// TwinCAT 3 PLC project Untitled1
// ProgramVersion: 3.1.4024.12
// libraries:
//   Tc2_Standard, * (Beckhoff Automation GmbH)
//   Tc2_System, * (Beckhoff Automation GmbH)
//   Tc3_Module, * (Beckhoff Automation GmbH)
// project tree:
//   Loadstation/ Parts.TcGVL, MAIN.TcPOU
//   Loadstation/State_Command_Enum/ Command.TcDUT, DUT.TcTLEO
//   / PlcTask.TcTTO
//   Loadstation/2_Control/ CON_LoadingStation.TcPOU
//   Loadstation/2_Control/Loadingstation/DataTypes/ MOD_Loadingstation_I_stWeighbridge.TcDUT (not stored), MOD_Loadingstation_Q_stCrane.TcDUT
//   Loadstation/3_Module/Crane/DataTypes/ MOD_Crane_I_stLoad.TcDUT, MOD_Crane_I_stSensor.TcDUT (not stored), MOD_Crane_Q_stMotor.TcDUT (not stored)
//   Loadstation/3_Module/Crane/ MOD_Crane.TcPOU
//   Loadstation/3_Module/InputBelt/DataTypes/ MOD_InputBelt_I_stSensor.TcDUT (not stored), MOD_InputBelt_Q_stMotor.TcDUT (not stored), MOD_InputBelt_Q_stOutput.TcDUT, MOD_InputBelt_Q_stRequest.TcDUT (not stored)
//   Loadstation/3_Module/InputBelt/ MOD_InputBelt.TcPOU
//   Loadstation/3_Module/ MOD_MechanicalGrabCrane.TcPOU (not stored)
//   Loadstation/3_Module/WeighBridge/DataTypes/ MOD_WeighBridge_I_stDefinitions.TcDUT, MOD_Weighbridge_I_stSensor.TcDUT (not stored), MOD_WeighBridge_Q_stOutput.TcDUT (not stored)
//   Loadstation/3_Module/WeighBridge/ MOD_Weighbridge.TcPOU
//   Loadstation/4_Devices/Motor_Notimplemented/Sensor/ DEV_Sensor_stOutput.TcDUT
//   Loadstation/4_Devices/ Motor_Notimplemented.TcPOU (not stored), Sensor_Notimplemented.TcPOU (not stored)
//   Loadstation/Application/ FB2_Control.TcPOU, FB3_Modules.TcPOU, FB4_Devices.TcPOU
// real-time tasks:
//   TASK PlcTask: cycle T#10ms, priority 20, ADS port 350

CONFIGURATION Untitled1
    RESOURCE PLC ON TwinCAT3
        TASK PlcTask(INTERVAL := T#10ms, PRIORITY := 20);
        PROGRAM MAIN WITH PlcTask : MAIN;
    END_RESOURCE
END_CONFIGURATION

// ---- Loadstation/State_Command_Enum/Command.TcDUT
{attribute 'qualified_only'}
{attribute 'strict'}
TYPE Command :
(
	Stop 		:= 0,
	Abort 		:= 1,
	Executing 	:= 2,
	Hold 		:= 3,
	Reset 		:= 4
);
END_TYPE

// ---- Loadstation/State_Command_Enum/DUT.TcTLEO
{attribute 'qualified_only'}
{attribute 'strict'}
TYPE DUT :
(
	Aborting := 0,
	Aborted		:= 1,
	
	Clearing	:= 2,
	Stopping	:= 3,
	Stopped		:= 4,
	
	Resetting	:= 5,
	Idle		:= 6,
	Starting	:= 7,
	Execute		:= 8,
	
	Holding		:= 9,
	Held		:= 10,
	Unholding		:= 11,
	
	Suspending		:= 12,
	Suspended		:= 13,
	Unsuspending	:= 14,
	
	Complete 		:= 15
);
END_TYPE

// ---- Loadstation/2_Control/Loadingstation/DataTypes/MOD_Loadingstation_Q_stCrane.TcDUT
TYPE MOD_Loadingstation_Q_stCrane :
STRUCT
	AllowedToOperate : BOOL;
END_STRUCT
END_TYPE

// ---- Loadstation/3_Module/Crane/DataTypes/MOD_Crane_I_stLoad.TcDUT
TYPE MOD_Crane_I_stLoad :
STRUCT
	Ready : BOOL;
	AllowedToOperate : BOOL;
END_STRUCT
END_TYPE

// ---- Loadstation/3_Module/InputBelt/DataTypes/MOD_InputBelt_Q_stOutput.TcDUT
TYPE MOD_InputBelt_Q_stOutput :
STRUCT
	BoxReady : BOOL;
END_STRUCT
END_TYPE

// ---- Loadstation/3_Module/WeighBridge/DataTypes/MOD_WeighBridge_I_stDefinitions.TcDUT
TYPE MOD_WeighBridge_I_stDefinitions :
STRUCT
	WeightLimit : INT;
	OperatingWeight : INT;
	DetractorWeight : INT;
END_STRUCT
END_TYPE

// ---- Loadstation/4_Devices/Motor_Notimplemented/Sensor/DEV_Sensor_stOutput.TcDUT
TYPE DEV_Sensor_stOutput :
STRUCT
	Abort : BOOL;
	Detecting : BOOL;
END_STRUCT
END_TYPE

// ---- Loadstation/Parts.TcGVL
//{attribute 'qualified_only'}
VAR_GLOBAL
	GlobalCommandState : INT;	

	//control
	Loadingstation : CON_LoadingStation; 
	
	//Modules
	Belt : MOD_InputBelt;
	Crane : MOD_Crane;
	Weighbridge : MOD_Weighbridge;
	MechanicalGrabCrane : MOD_MechanicalGrabCrane;
	
	//devices
END_VAR

// ---- Loadstation/MAIN.TcPOU
PROGRAM MAIN
VAR	
	Control : FB2_Control;
	Modules : FB3_Modules;
	
END_VAR

Control();
Modules();

END_PROGRAM

// ---- Loadstation/Application/FB2_Control.TcPOU
FUNCTION_BLOCK FB2_Control
VAR_INPUT
END_VAR
VAR_OUTPUT
END_VAR
VAR
END_VAR

//loadingstation
Loadingstation.i_weighbridge.TruckOnScale 			:= Weighbridge.q_Output.TruckOnScale;
Loadingstation.i_weighbridge.WeightLimitReached 	:= Weighbridge.q_Output.WeightLimitReached;

Loadingstation(iq_Commandstate := GlobalCommandState);

END_FUNCTION_BLOCK

// ---- Loadstation/Application/FB3_Modules.TcPOU
FUNCTION_BLOCK FB3_Modules
VAR_INPUT
END_VAR
VAR_OUTPUT
END_VAR
VAR
	newboxdump : MOD_InputBelt_Q_stRequest;
	WeighbridgeDefinitions : MOD_WeighBridge_I_stDefinitions;
END_VAR

//Belt
Belt(
	iq_Commandstate := Parts.GlobalCommandState,
	q_NewBox => newboxdump);

//weighbridge	
WeighbridgeDefinitions.DetractorWeight 	:= 60;// nust be set according to the max weight of delivered product.
WeighbridgeDefinitions.OperatingWeight 	:= 1000; // must be set to the minimum weight acceptable to respresent a truck. to prevent accidents.
WeighbridgeDefinitions.WeightLimit 		:= 6000; // needs to be set by external source like HMI	

Parts.Weighbridge(
	i_Definitions 		:= WeighbridgeDefinitions,
	iq_CommandState  	:= Parts.GlobalCommandState);

//crane
Crane.i_Input.Ready 	:= Belt.q_BoxReady.BoxReady;

Crane(
	i_LoadGrabbed 		:= Parts.MechanicalGrabCrane.q_Grabbed,
	q_Grab 				=> Parts.MechanicalGrabCrane.i_Grab,
	iq_CommandState 	:= Parts.GlobalCommandState);

//grabcrane	
Parts.MechanicalGrabCrane(iq_CommandState  := Parts.GlobalCommandState);

END_FUNCTION_BLOCK

// ---- Loadstation/2_Control/CON_LoadingStation.TcPOU
FUNCTION_BLOCK CON_LoadingStation
VAR_INPUT
	i_weighbridge 					: MOD_Loadingstation_I_stWeighbridge;
	i_tempIWantExtraBoxInTruck 		: BOOL;
END_VAR
VAR_OUTPUT
	q_crane 						: MOD_Loadingstation_Q_stCrane;
END_VAR
VAR_IN_OUT
	iq_CommandState 				: INT;
END_VAR
VAR
	resetTimer						: TON;
	resetState 						: INT;
END_VAR

//check if there is a truck before running. Also check for weightlimit
IF NOT i_weighbridge.TruckOnScale THEN
	q_crane.AllowedToOperate 	:= FALSE;
	iq_CommandState 			:= Command.Abort;
	//Abort no truck
ELSIF i_weighbridge.TruckOnScale AND NOT i_weighbridge.WeightLimitReached THEN
	q_crane.AllowedToOperate 	:= TRUE;//can come fromoutside?
	CASE resetState OF
		0:
			iq_CommandState 	:= Command.Reset;
			resetTimer(IN := TRUE, PT := T#2S);
			IF resetTimer.Q THEN
				resetTimer(IN := FALSE, PT := T#2S);
				resetState := 1;				
			END_IF
		1:
			iq_CommandState 	:= Command.Executing;
	END_CASE
// if operator wants an extra box loaded above the limit.
ELSIF i_tempIWantExtraBoxInTruck THEN //is supposed to be a button press
	q_crane.AllowedToOperate 	:= TRUE;
	CASE resetState OF
		0:
			iq_CommandState 	:= Command.Reset;
			resetTimer(IN := TRUE, PT := T#2S);
			IF resetTimer.Q THEN
				resetTimer(IN := FALSE, PT := T#2S);
				resetState := 1;				
			END_IF

		1:
			iq_CommandState 	:= Command.Executing;
	END_CASE
ELSIF i_weighbridge.WeightLimitReached THEN
	q_crane.AllowedToOperate 	:= FALSE;
	iq_CommandState 			:= Command.Stop;
	//done loading!
END_IF



CASE iq_CommandState OF
	Command.Abort:
		resetState := 0;
	Command.Reset:
		resetState := 0;
END_CASE

END_FUNCTION_BLOCK

// ---- Loadstation/3_Module/InputBelt/MOD_InputBelt.TcPOU
FUNCTION_BLOCK MOD_InputBelt
VAR_INPUT
	i_InputSensor 	: MOD_InputBelt_I_stSensor;
	i_OutputSensor 	: MOD_InputBelt_I_stSensor;
END_VAR
VAR_OUTPUT
	q_NewBox 		: MOD_InputBelt_Q_stRequest;
	q_BeltMotorOn 	: MOD_InputBelt_Q_stMotor := (MoveLeft := FALSE, MoveRight := FALSE);
	q_BoxReady 		: MOD_InputBelt_Q_stOutput;
END_VAR
VAR_IN_OUT
	iq_CommandState : INT;
END_VAR
VAR
	State 			: INT := 10;
	Executing 		: BOOL := FALSE;//variable for main state. used for orderly code
END_VAR

CASE iq_CommandState OF
	Command.Abort:
		q_BeltMotorOn.MoveLeft 	:= FALSE;
		Executing 				:= FALSE;
		
	Command.Executing:
		Executing 				:= TRUE;
		
	Command.Hold:
		Executing 				:= FALSE;
		q_BeltMotorOn.MoveLeft 	:= FALSE;
		
	Command.Reset:
		Executing 				:= FALSE;
		State 					:= 10;//reset state
		q_BeltMotorOn.MoveLeft 	:= FALSE;
		
	Command.Stop:		
		IF State = 20 THEN
			Executing 				:= FALSE;
			q_BeltMotorOn.MoveLeft 	:= FALSE;
		ELSE
			Executing 				:= TRUE;			
		END_IF		
END_CASE

IF Executing THEN
CASE State OF
	10://startup //reset?
		IF i_InputSensor.Blocked = TRUE AND i_OutputSensor.Blocked = TRUE THEN
			State := 11;
		ELSIF i_InputSensor.Blocked = FALSE AND i_OutputSensor.Blocked = FALSE THEN
			State := 20;
		ELSIF i_InputSensor.Blocked = TRUE AND i_OutputSensor.Blocked = FALSE THEN
			State := 30;
		ELSIF i_InputSensor.Blocked = FALSE AND i_OutputSensor.Blocked = TRUE THEN
			State := 40;		
		END_IF
		
	11://startup boxes on belt.
		q_NewBox.NewBox 		:= FALSE;
		q_BeltMotorOn.MoveLeft 	:= FALSE;
		q_BoxReady.BoxReady 	:= TRUE;
	
		IF i_OutputSensor.Blocked = FALSE THEN
			State := 20;
		END_IF
		
	20://No Box
		q_NewBox.NewBox 		:= TRUE;
		q_BeltMotorOn.MoveLeft 	:= FALSE;
		q_BoxReady.BoxReady 	:= FALSE;
		
		IF i_InputSensor.Blocked = TRUE AND i_OutputSensor.Blocked = FALSE THEN
			State := 30;
		END_IF
	
	30://retrieve box
		q_NewBox.NewBox 		:= FALSE;
		q_BeltMotorOn.MoveLeft 	:= TRUE;
		q_BoxReady.BoxReady 	:= FALSE;
		
		IF i_InputSensor.Blocked = FALSE AND i_OutputSensor.Blocked = TRUE THEN
			State := 40;
		END_IF
		
	40://boxready
		q_NewBox.NewBox 		:= FALSE;
		q_BeltMotorOn.MoveLeft 	:= FALSE;
		q_BoxReady.BoxReady 	:= TRUE;
		
		IF i_OutputSensor.Blocked = FALSE THEN
			State := 20;
		END_IF

END_CASE
END_IF

END_FUNCTION_BLOCK

// ---- Loadstation/3_Module/Crane/MOD_Crane.TcPOU
FUNCTION_BLOCK MOD_Crane
VAR_INPUT
	i_CraneDownSensor 	: MOD_Crane_I_stSensor;
	i_CraneUpSensor 	: MOD_Crane_I_stSensor;
	i_CraneAbovePickupSensor 	: MOD_Crane_I_stSensor;
	i_CraneAboveDropoffSensor 	: MOD_Crane_I_stSensor;

	i_Input 			: MOD_Crane_I_stLoad;
	i_LoadGrabbed 		: BOOL;
END_VAR
VAR_OUTPUT
	//right is down left is up
	q_HorizontalMotor 	: MOD_Crane_Q_stMotor;
	q_VerticalMotor 	: MOD_Crane_Q_stMotor;
	q_Grab 				: BOOL;
END_VAR
VAR_IN_OUT
	iq_CommandState 	: INT;
END_VAR
VAR
	State				: INT := 10;
	MotorDirection 		: (Left, Right, Stopped);
	Executing 			: BOOL := FALSE;//variable for main state. used for orderly code		
END_VAR

CASE iq_CommandState OF
	Command.Abort:
		Executing 					:= FALSE;
		q_VerticalMotor.MoveLeft 	:= FALSE;
		q_VerticalMotor.MoveRight 	:= FALSE;
		q_HorizontalMotor.MoveLeft 	:= FALSE;
		q_HorizontalMotor.MoveRight := FALSE;
		
	Command.Executing:
		Executing 					:= TRUE;
		
	Command.Hold:
		Executing 					:= FALSE;
		q_VerticalMotor.MoveLeft 	:= FALSE;
		q_VerticalMotor.MoveRight 	:= FALSE;
		q_HorizontalMotor.MoveLeft 	:= FALSE;
		q_HorizontalMotor.MoveRight := FALSE;
		
	Command.Reset:
		Executing 					:= FALSE;
		State 						:= 10;//reset state
		q_VerticalMotor.MoveLeft 	:= FALSE;
		q_VerticalMotor.MoveRight 	:= FALSE;
		q_HorizontalMotor.MoveLeft 	:= FALSE;
		q_HorizontalMotor.MoveRight := FALSE;
		
	Command.Stop:
		IF State = 20 THEN
			Executing 					:= FALSE;
			q_VerticalMotor.MoveLeft 	:= FALSE;
			q_VerticalMotor.MoveRight 	:= FALSE;
			q_HorizontalMotor.MoveLeft 	:= FALSE;
			q_HorizontalMotor.MoveRight := FALSE;	
		ELSE
			Executing 					:= TRUE;	
		END_IF
END_CASE


IF Executing THEN
CASE State OF
	10://startup //reset?
		q_VerticalMotor.MoveLeft 	:= FALSE;
		q_VerticalMotor.MoveRight 	:= FALSE;
		q_HorizontalMotor.MoveLeft 	:= FALSE;
		q_HorizontalMotor.MoveRight := FALSE;
		
		IF i_CraneAbovePickupSensor.Blocked THEN
			State := 20;
		ELSE
			State := 90;
		END_IF
		
	20://operational approval
		q_VerticalMotor.MoveLeft 	:= FALSE;
		q_VerticalMotor.MoveRight 	:= FALSE;
		q_HorizontalMotor.MoveLeft 	:= FALSE;
		q_HorizontalMotor.MoveRight := FALSE;
		//wait untill
		IF i_Input.AllowedToOperate = TRUE THEN
			State := 21;
		END_IF
		
	21://check box ready
		q_VerticalMotor.MoveLeft 	:= FALSE;
		q_VerticalMotor.MoveRight 	:= FALSE;
		q_HorizontalMotor.MoveLeft 	:= FALSE;
		q_HorizontalMotor.MoveRight := FALSE;
		//wait untill
		IF i_Input.Ready = TRUE THEN
			State := 30;
		END_IF
	
	30://move crane down
		
		q_VerticalMotor.MoveLeft 	:= TRUE;
		q_VerticalMotor.MoveRight 	:= FALSE;
		q_HorizontalMotor.MoveLeft 	:= FALSE;
		q_HorizontalMotor.MoveRight := FALSE;
		
		IF i_CraneDownSensor.Blocked = TRUE THEN
			State := 40;
		END_IF
		
	40://grab the load
		q_VerticalMotor.MoveLeft 	:= FALSE;
		q_VerticalMotor.MoveRight 	:= FALSE;
		q_HorizontalMotor.MoveLeft 	:= FALSE;
		q_HorizontalMotor.MoveRight := FALSE;
		
		q_Grab 						:= TRUE;
		
		IF i_LoadGrabbed = TRUE THEN
			State := 50;
		END_IF

	50://move crane up
		q_VerticalMotor.MoveLeft 	:= TRUE;
		q_VerticalMotor.MoveRight 	:= FALSE;
		q_HorizontalMotor.MoveLeft 	:= FALSE;
		q_HorizontalMotor.MoveRight := FALSE;
		
		q_Grab 						:= TRUE;
		
		IF i_CraneUpSensor.Blocked = TRUE THEN
			State := 60;
		END_IF

	60://move crane to output position
		q_VerticalMotor.MoveLeft 	:= FALSE;
		q_VerticalMotor.MoveRight 	:= FALSE;
		q_HorizontalMotor.MoveLeft 	:= TRUE;
		q_HorizontalMotor.MoveRight := FALSE;
		
		q_Grab 						:= TRUE;
		
		IF i_CraneAboveDropoffSensor.Blocked = TRUE THEN
			State := 70;
		END_IF

	70://move crane down
		q_VerticalMotor.MoveLeft 	:= FALSE;
		q_VerticalMotor.MoveRight 	:= TRUE;
		q_HorizontalMotor.MoveLeft 	:= FALSE;
		q_HorizontalMotor.MoveRight := FALSE;	
	
		IF i_CraneDownSensor.Blocked = TRUE THEN
			State := 80;
		END_IF

	80://release load
		q_Grab := FALSE;
		IF i_LoadGrabbed = FALSE THEN
			State := 90;
		END_IF

	90://move crane up
		q_VerticalMotor.MoveLeft 	:= TRUE;
		q_VerticalMotor.MoveRight 	:= FALSE;
		q_HorizontalMotor.MoveLeft 	:= FALSE;
		q_HorizontalMotor.MoveRight := FALSE;	
		
		IF i_CraneUpSensor.Blocked = TRUE THEN
			State := 100;
		END_IF	

	100://move crane over input
		q_VerticalMotor.MoveLeft 	:= FALSE;
		q_VerticalMotor.MoveRight 	:= FALSE;
		q_HorizontalMotor.MoveLeft 	:= FALSE;
		q_HorizontalMotor.MoveRight := TRUE;
		
		IF i_CraneAbovePickupSensor.Blocked = TRUE THEN
			State := 20;
		END_IF
END_CASE
END_IF

END_FUNCTION_BLOCK

// ---- Loadstation/3_Module/WeighBridge/MOD_Weighbridge.TcPOU
FUNCTION_BLOCK MOD_Weighbridge
VAR_INPUT
	i_Definitions 	: MOD_WeighBridge_I_stDefinitions;
	i_Sensor 		: MOD_Weighbridge_I_stSensor;
END_VAR
VAR_OUTPUT
	q_Output 		: MOD_WeighBridge_Q_stOutput;
END_VAR
VAR_IN_OUT
	iq_CommandState : INT;
END_VAR
VAR
	State 			: INT;
END_VAR

IF iq_CommandState = Command.Executing OR iq_CommandState = Command.Hold THEN

	q_Output.TruckOnScale := i_Sensor.Weight > i_Definitions.OperatingWeight;

	q_Output.WeightLimitReached := i_Definitions.WeightLimit - i_Definitions.DetractorWeight < i_Sensor.Weight;
	
ELSE
	q_Output.TruckOnScale := FALSE;
	q_Output.WeightLimitReached := FALSE;
END_IF

END_FUNCTION_BLOCK

// ---- Loadstation/Application/FB4_Devices.TcPOU
FUNCTION_BLOCK FB4_Devices
VAR_INPUT
END_VAR
VAR_OUTPUT
END_VAR
VAR
END_VAR

//devices are not implemented for this project

END_FUNCTION_BLOCK
